// TIA Portal project "LVT_ModbusDeviceRtu_slow-poll_v0.0.1" (V17)

(* hardware
DEVICE "S7-1200 station_1"  S7-1200 Station
   slot 0: "Rack_0"  S7-1200 Rack  Rack  V1.0
   slot 1: "PLC_1"  CPU 1214C DC/DC/DC  6ES7 214-1AG40-0XB0  V4.3
   slot 3: "CB1"  CB 1241 (RS485)  6ES7 241-1CH30-1XB0  V1.0
*)

// ===== PLC "PLC_1"  CPU 1214C DC/DC/DC =====

VAR_GLOBAL   // PLC tag table "Default tag table"
   "System_Byte" AT %MB500 : Byte;
   "FirstScan" AT %M500.0 : Bool;
   "DiagStatusUpdate" AT %M500.1 : Bool;
   "AlwaysTRUE" AT %M500.2 : Bool;
   "AlwaysFALSE" AT %M500.3 : Bool;
   "System_Byte(1)" AT %MB1 : Byte;
   "System_Byte(2)" AT %MB1 : Byte;
   "Clock_Byte" AT %MB501 : Byte;
   "Clock_10Hz" AT %M501.0 : Bool;
   "Clock_5Hz" AT %M501.1 : Bool;
   "Clock_2.5Hz" AT %M501.2 : Bool;
   "Clock_2Hz" AT %M501.3 : Bool;
   "Clock_1.25Hz" AT %M501.4 : Bool;
   "Clock_1Hz" AT %M501.5 : Bool;
   "Clock_0.625Hz" AT %M501.6 : Bool;
   "Clock_0.5Hz" AT %M501.7 : Bool;
END_VAR

// folder: Example

TYPE "DeviceData"
   STRUCT
      param1 : Word;   // Parameter 1
      error : Bool;   // Flag. The device don't respond
   END_STRUCT;
END_TYPE

// folder: LVT_ModbusDeviceRtu

TYPE "LVT_typeModbusDeviceRtu_RequestCfg"
// Modbus request configuration
   STRUCT
      mode : USInt := 0;   // Mode / Режим опроса
      dataAddr : UDInt := 40001;   // Starting address in the slave / Начальный адрес регистра
      len : UInt := 1;   // Data length / Длина запроса
      mapAddr : DInt := 0;   // Starting address in the read/write buffer
      enable : Bool := false;   // Заблокировать запрос / Enable request
   END_STRUCT;
END_TYPE

TYPE "LVT_typeModbusDeviceRtu_Request"
   STRUCT
      cfg : "LVT_typeModbusDeviceRtu_RequestCfg";
      status : "LVT_typeModbusDeviceRtu_RequestStatus";
   END_STRUCT;
END_TYPE

TYPE "LVT_typeModbusDeviceRtu_Data"
   STRUCT
      address : UInt;   // Modbus RTU station address
      buffer : Array[0..100] of Word;   // Local buffer
      requests : Array[0..9] of "LVT_typeModbusDeviceRtu_Request";   // Requests
   END_STRUCT;
END_TYPE

TYPE "LVT_typeModbusDeviceRtu_RequestStatus"
// Modbus request status
   STRUCT
      req : Bool;   // Команда на отпарвку запроса / Send request
      done : Bool;   // Опрос завершен / Request is done
      busy : Bool;   // Блок в работе / Request is in progress
      error : Bool;   // Ошибка / Error
      status : Word;   // Статус / Error code
      errorCounter : UInt;   // Counter of failed attempts
   END_STRUCT;
END_TYPE

TYPE "LVT_typeModbusDeviceRtu_ComPortData"
TITLE = Настройки COM-порта
// Настройки COM-порта
   STRUCT
      port : Port := 271;   // ID порта / ID Port
      baud : UDInt := 9600;   // Скорость / Baudrate
      parity : UInt := 2;   // Паритет (0 - Нет, 1 - Нечет, 2 - Чет ) / Parity (0- None, 1 - Odd, 2 - Even)
      stopBits : UInt;   // Number of stop bits per character Valid values 1 and 2
      timeout : UInt := 500;   // Максимальное время ответа / Response timeout, ms
      retries : Word := 2;   // Количество повторных запросово / The number of repeated attempts by the master before the error code 0x80C8 is returned for "No response
      status : Word;   // Статус / Error codes
      done : Bool;   // Инициализация завершена / Execution of instruction completed without error
      error : Bool;   // Ошибка инициализации / Error
   END_STRUCT;
END_TYPE

// folder: Example/Data

DATA_BLOCK "DataDb"   // DB1
{ S7_Optimized_Access := 'TRUE' }
VERSION : 0.1
   VAR
      devices : Array[0..2] of "DeviceData";
   END_VAR
BEGIN
END_DATA_BLOCK

DATA_BLOCK "ModbusRtuMaster_DevicesDb"   // DB2
{ S7_Optimized_Access := 'TRUE' }
VERSION : 0.1
   VAR RETAIN
      devices : Array[0..2] of "LVT_typeModbusDeviceRtu_Data";
   END_VAR
BEGIN
   devices[0].address := 1;
   devices[1].address := 2;
   devices[2].address := 3;
   devices[0].requests[0].cfg.mode := 0;
   devices[0].requests[0].cfg.dataAddr := 40001;
   devices[0].requests[0].cfg.len := 1;
   devices[0].requests[0].cfg.mapAddr := 0;
   devices[0].requests[0].cfg.enable := true;
   devices[1].requests[0].cfg.mode := 0;
   devices[1].requests[0].cfg.dataAddr := 40001;
   devices[1].requests[0].cfg.len := 1;
   devices[1].requests[0].cfg.mapAddr := 0;
   devices[1].requests[0].cfg.enable := true;
   devices[2].requests[0].cfg.mode := 0;
   devices[2].requests[0].cfg.dataAddr := 40001;
   devices[2].requests[0].cfg.len := 1;
   devices[2].requests[0].cfg.mapAddr := 0;
   devices[2].requests[0].cfg.enable := true;
END_DATA_BLOCK

DATA_BLOCK "LVT_ModbusDeviceRtu_CfgDb"   // DB21
{ S7_Optimized_Access := 'TRUE' }
AUTHOR : Veshtemov
VERSION : 0.1
// Конфигурация регистров чтения по Modbus RTU
   VAR RETAIN
      com : "LVT_typeModbusDeviceRtu_ComPortData";
   END_VAR
BEGIN
   com.retries := 1;
   com.timeout := 500;
   com.port := 271;
   com.baud := 9600;
   com.parity := 0;
   com.stopBits := 0;
END_DATA_BLOCK

DATA_BLOCK "LVT_ModbusDeviceRtu_DataDb"   // DB24
{ S7_Optimized_Access := 'FALSE' }
VERSION : 0.1
   VAR
      readBuffer : Array[0..255] of Byte;
      writeBuffer : Array[0..255] of Byte;
   END_VAR
BEGIN
END_DATA_BLOCK

// folder: Example/Inst

DATA_BLOCK "inst_ModbusRtu_Master"   // DB3
{ S7_Optimized_Access := 'TRUE' }
VERSION : 0.1
// stored: InstanceOfName ModbusRtu_Master
"ModbusRtu_Master"
BEGIN
END_DATA_BLOCK

// folder: Example

ORGANIZATION_BLOCK "Main"   // OB1, SCL, ProgramCycle
TITLE = "Main Program Sweep (Cycle)"
{ S7_Optimized_Access := 'TRUE' }
VERSION : 0.1
   VAR_INPUT
      Initial_Call : Bool;   // Initial call of this OB
      Remanence : Bool;   // =True, if remanent data are available
   END_VAR
BEGIN
   "inst_ModbusRtu_Master"(com:="LVT_ModbusDeviceRtu_CfgDb".com,
                           mbCommLoad:="Modbus_Comm_Load_DB",
                           mbMaster:="Modbus_Master_DB");
END_ORGANIZATION_BLOCK

// folder: Example/RS485/ModbusRtuMaster

FUNCTION_BLOCK "ModbusRtu_Master"   // FB5, SCL
{ S7_Optimized_Access := 'TRUE' }
VERSION : 0.1
// Modbus Rtu Bus
   VAR_IN_OUT
      com : "LVT_typeModbusDeviceRtu_ComPortData";   // Serial port settings
      mbCommLoad : Modbus_Comm_Load;   // Instance of "Modbus_Comm_Load" function block
      mbMaster : Modbus_Master;   // Instance of "Modbus_Master" function block
   END_VAR
   VAR
      allowPolles : Array[0..#MAX_DEV_INDEX] of Bool;   // Allow polling
      slowPollTimers : Array[0..#MAX_DEV_INDEX] of TON_TIME;   // Slow poll timer
      stat_InitTrig : R_TRIG;   // Trig to set serial port is ready
      stat_LModbusDeviceRtu_Master : "LVT_ModbusDeviceRtu_Master";   // Instance of "LMBMD_ModbusDevice"
      i : Int := 0;   // Index
      j : Int := 0;   // Index
      statStart : Bool;   // Flag to start polling
   END_VAR
   VAR CONSTANT
      MAX_DEV_INDEX : Int := 2;   // Max index in devices array
      SLOW_POLL_TIME : Time := T#10s;   // Slow poll time
   END_VAR
BEGIN
   REGION Block info header
       //===============================================================================
       // (company) / (c)Copyright year
       //-------------------------------------------------------------------------------
       // Title:            Example of LVT _ModbusDevcieRtu library
       // Comment/Function: Modbus RTU Master device-oriented
       //                   This functional block polls 1 register in 3 indentical devices,
       //                   If a device fails to respond 3 times, a slowPollTimer is activated 
       //                   and polling is blocked until timer expires
       // Library/Family:   LMB (Library Modbus)
       // Author:           Anatoly Veshtemov
       // Tested with:      CPU 1214C
       // Engineering:      TIA Portal V17
       // Restrictions:     no
       // Requirements:     PLC (S7-1200 / S7-1500)
       //-------------------------------------------------------------------------------
       // Change log table:
       // Version  | Date       | Expert in charge       | Changes applied
       //----------|------------|------------------------|------------------------------
       // 00.01.00 17.06.2026  First release
       //=============================================================================

   END_REGION Block info header

   REGION DESCRIPTION
       (/**/)
   END_REGION DESCRIPTION


   // Modbus RTU Master

   REGION Serial port initialization
       IF "FirstScan" THEN
           #mbCommLoad.MODE := 4;
       END_IF;

       #mbCommLoad.RETRIES := #com.retries;

       #mbCommLoad(REQ := "FirstScan",
                   "PORT" := #com."port",
                   BAUD := #com.baud,
                   PARITY := #com.parity,
                   MB_DB := #mbMaster.MB_DB,
                   RESP_TO := #com.timeout,
                   DONE => #com.done,
                   ERROR => #com.error,
                   STATUS => #com.status);

       #stat_InitTrig(CLK := #com.done);

       IF #stat_InitTrig.Q THEN
           #i := 0;
       END_IF;
   END_REGION

   #statStart := NOT #stat_LModbusDeviceRtu_Master.done;

   REGION Slow poll

       FOR #j := 0 TO #MAX_DEV_INDEX DO

           // Update Slow Poll timers
           #slowPollTimers[#j](IN := "DataDb".devices[#j].error,
                               PT := #SLOW_POLL_TIME);

           // Polling is allowed if there are no error or timer is ended.        
           #allowPolles[#j] := NOT ("DataDb".devices[#j].error AND #slowPollTimers[#j].Q);

       END_FOR;

   END_REGION

   CASE #i OF
       0..#MAX_DEV_INDEX:  // Device 1..Devices 3

           IF #allowPolles[#i] THEN
               #stat_LModbusDeviceRtu_Master(start := #statStart,
                                             readBuffer := "LVT_ModbusDeviceRtu_DataDb".readBuffer,
                                             writeBuffer := "LVT_ModbusDeviceRtu_DataDb".writeBuffer,
                                             data := "ModbusRtuMaster_DevicesDb".devices[#i],
                                             mbMaster := #mbMaster);

               IF #stat_LModbusDeviceRtu_Master.done THEN

                   "ModbusRtu_Device_HandleData"(mdata := "ModbusRtuMaster_DevicesDb".devices[#i],
                                                 data := "DataDb".devices[#i]);

                   #i := #i + 1;
               END_IF;

           ELSE
               #i := #i + 1;
           END_IF;

       ELSE
           #i := 0;
   END_CASE;
END_FUNCTION_BLOCK

FUNCTION "ModbusRtu_Device_HandleData" : Void   // FC18, SCL
{ S7_Optimized_Access := 'TRUE' }
VERSION : 0.1
   VAR_IN_OUT
      mdata : "LVT_typeModbusDeviceRtu_Data";
      data : "DeviceData";
   END_VAR
   VAR_TEMP
      i : Int;   // Increment
      statQuantityErrors : UInt;   // Quantity of failed requests
   END_VAR
   VAR CONSTANT
      ERRORS_THRESHOLD : Int := 3;   // Max. quantity of failed requests
      MAX_REQUEST_INDEX : Int := 9;   // Max. index of array with requests
   END_VAR
BEGIN
   REGION Block info header
       //===============================================================================
       // (company) / (c)Copyright year
       //-------------------------------------------------------------------------------
       // Title:            Example of LVT_ModbusDevcieRtu library
       // Comment/Function: Modbus RTU Master device-oriented
       //                   Copy data to device from modbus buffer, set connection status
       // Library/Family:   LVT 
       // Author:           Anatoly Veshtemov
       // Tested with:      CPU 1214C
       // Engineering:      TIA Portal V17
       // Restrictions:     no
       // Requirements:     PLC (S7-1200 / S7-1500)
       //-------------------------------------------------------------------------------
       // Change log table:
       // Version  | Date       | Expert in charge       | Changes applied
       //----------|------------|------------------------|------------------------------
       // 00.00.01 17.06.2026  First release
       //=============================================================================

   END_REGION Block info header

   REGION DESCRIPTION
       (/**/)
   END_REGION DESCRIPTION


   // Data
   #data.param1 := #mdata.buffer[0];

   // Calculate quantity of failed requests
   #statQuantityErrors := 0;
   FOR #i := 0 TO #MAX_REQUEST_INDEX - 1 DO
       #statQuantityErrors += #mdata.requests[#i].status.errorCounter;
   END_FOR;

   // Set error status
   #data.error := #statQuantityErrors >= #ERRORS_THRESHOLD;
END_FUNCTION

// folder: LVT_ModbusDeviceRtu

FUNCTION "LVT_ModbusDeviceRtu_Description" : Void   // FC3, SCL
{ S7_Optimized_Access := 'TRUE' }
AUTHOR : Anatoly Veshtemov
FAMILY : LVT
BEGIN
   REGION INFO
   (/*title: Library for Modbus Rtu Master
   subTitle: STEP 7 Basic/Professional (TIA PORTAL) / SIMATIC S7-1200 / S7-1500
   shortDescription: Modbus RTU Master device-oriented library for S7-1200/S7-1500
   type: Library
   fileName: LVT_ModbusDeviceRtu_Lib
   link: https://github.com/vapik/simatic-modbus-device-master*/)
   END_REGION INFO

   REGION ChangeLog
   (*
   Version  | Date       | Expert in charge       | Changes applied
   ---------|------------|------------------------|------------------------------
   00.01.00 | 17.06.2026 | Upgrate to TIA V17
            |            | Added block info headers
            |            | Refactor names
            |            | Examples has deleted                  
            |            | Chanhed name to LVT_ModbusDeviceRtu                           
   *)
   END_REGION
END_FUNCTION

// folder: LVT_ModbusDeviceRtu/Core

FUNCTION_BLOCK "LVT_ModbusDeviceRtu_Master"   // FB7, SCL
{ S7_Optimized_Access := 'TRUE' }
AUTHOR : Anatoly Veshtemov
FAMILY : LVT
   VAR_INPUT
      start : Bool;   // Пуск / Start block
   END_VAR
   VAR_OUTPUT
      busy : Bool;   // В процессе / In progress
      done : Bool;   // Окончание / Done
   END_VAR
   VAR_IN_OUT
      readBuffer : Variant;   // Буфер обмена / Pointer of read buffer (non optimized data block). For example, DB -> readBuffer: Array[0..125] of Word
      writeBuffer : Variant;   // Pointer of write buffer (non optimized data block). For example, DB -> writeBuffer: Array[0..125] of Word
      data : "LVT_typeModbusDeviceRtu_Data";
      mbMaster : Modbus_Master;   // Instance of Modbus_Master function block
   END_VAR
   VAR
      statBuffer : Array[0..127] of Word;
      startTrig : R_TRIG;   // Detect start
      statWatchdogTimer : TON_TIME;   // Timer for resetting a request when unknown reason is happened
      statState : USInt;   // Текущая стадия обмена / Current state
      i : Int;
      j : Int;
   END_VAR
   VAR_TEMP
      tempStart : Bool;   // Start flag
      tempRetval : Int;
      tempQntRequests : Int;   // Quantity of requests
      tempZeroIndex : DInt;
   END_VAR
   VAR CONSTANT
      STATE_STANDBY : USInt := 0;   // Ожидание / State. Standby
      STATE_SETTINGS : USInt := 1;   // Конфигурирование запроса / State. Get settings
      STATE_READ : USInt := 2;   // Запрос на чтение / State. Reading
      STATE_WRITE : USInt := 3;   // Запрос на запись / State. Writing
      STATE_HANDLE : USInt := 4;   // Обработка запроса / State. Handle results
      WATCHDOG_TIME : Time := T#10S;   // Максимальное время ожидания / Watchdog time
      ERROR_ILLEGAL_REQUEST : Word := 16#9000;   // Error. Illegal request (check request settings)
      ERROR_WATCHDOG_TIMER : Word := 16#9001;   // Error. Watchdog timer
   END_VAR
BEGIN
   REGION Block info header
       //===============================================================================
       // (company) / (c)Copyright year
       //-------------------------------------------------------------------------------
       // Title:            LVT_ModbusDevcieRtu_Master
       // Comment/Function: Modbus RTU Master device-oriented
       //                   Requests are grouped for each network device separately, and devices are sequentially polled.
       //                   Each network device has a local data buffer.
       // Library/Family:   LVT
       // Author:           Anatoly Veshtemov
       // Tested with:      CPU 1214C
       // Engineering:      TIA Portal V17
       // Restrictions:     no
       // Requirements:     PLC (S7-1200 / S7-1500)
       //-------------------------------------------------------------------------------
       // Change log table:
       // Version  | Date       | Expert in charge       | Changes applied
       //----------|------------|------------------------|------------------------------
       // 00.00.04 01.01.2023  First released version
       // 00.01.00 17.06.2026  Upgrate to TIA V17
       //                      Added block info header
       //                      Refactor names in Static 
       //=============================================================================

   END_REGION Block info header

   REGION DESCRIPTION
       (/**/)
   END_REGION DESCRIPTION

   #tempQntRequests := UDINT_TO_INT("LVT_ModbusDeviceRtu_GetArrayLength"(arr := #data.requests));
   #busy := (#statState > #STATE_STANDBY); // Set busy flag

   #startTrig(CLK := #start,
                   Q => #tempStart);

   // When start go to Settings
   IF #tempStart THEN

       #done := false;
       #statState := #STATE_SETTINGS;

   END_IF;

   CASE #statState OF

           // Standby
       #STATE_STANDBY:

           #done := false;
           #i := 0;

           // Get request settings
       #STATE_SETTINGS:

           // With the first call we reset the counter, get the first request,
           // else we increase counter by 1 and get a next request
           IF #tempStart THEN
               #i := 0;

           ELSE
               #i := #i + 1;

               // When all requests is completed go to standby, set "done" flag 
               IF #i >= #tempQntRequests THEN
                   #done := true;
                   #statState := #STATE_STANDBY;
                   RETURN;
               END_IF;
           END_IF;

           // Check request settings: we have to skip disabled or invalid requests,
           // if a request is invalid - set ERROR_ILLEGAL_REQUEST status
           FOR #j := #i TO #tempQntRequests - 1 DO

               IF NOT #data.requests[#j].cfg.enable THEN

                   #data.requests[#j].status.req := false;
                   #data.requests[#j].status.done := false;
                   #data.requests[#j].status.error := false;
                   #data.requests[#j].status.status := 0;
                   #data.requests[#j].status.errorCounter := 0;

               ELSIF NOT "LVT_ModbusDeviceRtu_ValidateRequest"(data := #data, index := #j) THEN

                   // Set error status
                   #data.requests[#j].status.req := false;
                   #data.requests[#j].status.done := false;
                   #data.requests[#j].status.error := true;
                   #data.requests[#j].status.status := #ERROR_ILLEGAL_REQUEST;
                   #data.requests[#j].status.errorCounter := LIMIT(IN := #data.requests[#j].status.errorCounter + 1,
                                                                   MN := 0,
                                                                   MX := 65534);
               ELSE
                   #i := #j;
                   EXIT;
               END_IF;

               // When all requests is completed go to standby, set "done" flag
               IF #j = #tempQntRequests - 1 THEN
                   #done := true;
                   #statState := #STATE_STANDBY;
                   RETURN;
               END_IF;

           END_FOR;

           // For writing before request we have to copy data to external write buffer
           IF #data.requests[#i].cfg.mode > 0 THEN

               // Extract data from Modbus Device to write buffer
               MOVE_BLK(IN := #data.#buffer[#data.requests[#i].cfg.mapAddr],
                        COUNT := #data.requests[#i].cfg.len,
                        OUT => #statBuffer[0]);

               #tempZeroIndex := 0;
               #tempRetval := Serialize(SRC_VARIABLE := #statBuffer,
                                        DEST_ARRAY => #writeBuffer,
                                        POS := #tempZeroIndex);

               #statState := #STATE_WRITE;
           ELSE
               #statState := #STATE_READ;
           END_IF;

           RETURN;

           // Read
       #STATE_READ, #STATE_WRITE:

           #data.requests[#i].status.req := true;

           // Handle results
       #STATE_HANDLE:

           #data.requests[#i].status.req := false;

           IF #data.requests[#i].status.done THEN
               #data.requests[#i].status.errorCounter := 0;

               // Copy from modbus buffer to device buffer
               IF #data.requests[#i].cfg.mode = 0 THEN

                   #tempZeroIndex := 0;
                   #tempRetval := Deserialize(SRC_ARRAY := #readBuffer,
                                              DEST_VARIABLE => #statBuffer,
                                              POS := #tempZeroIndex);
                   MOVE_BLK(IN := #statBuffer[0],
                            COUNT := #data.requests[#i].cfg.len,
                            OUT => #data.buffer[#data.requests[#i].cfg.mapAddr]);
               END_IF;

           ELSIF #data.requests[#i].status.error THEN
               #data.requests[#i].status.errorCounter := LIMIT(IN := #data.requests[#i].status.errorCounter + 1,
                                                               MN := 0,
                                                               MX := 65534);
           END_IF;

           #statState := #STATE_SETTINGS;

       ELSE
           #statState := #STATE_STANDBY;
   END_CASE;

   // There are different buffers for reading and writing
   IF (#statState = #STATE_READ) THEN
       // Request
       #mbMaster(REQ := #data.requests[#i].status.req,
                 MB_ADDR := #data.address,
                 MODE := #data.requests[#i].cfg.mode,
                 DATA_ADDR := #data.requests[#i].cfg.dataAddr,
                 DATA_LEN := #data.requests[#i].cfg.len,
                 DONE => #data.requests[#i].status.done,
                 BUSY => #data.requests[#i].status.busy,
                 ERROR => #data.requests[#i].status.error,
                 STATUS => #data.requests[#i].status.status,
                 DATA_PTR := #readBuffer);

   ELSIF (#statState = #STATE_WRITE) THEN
       // Request
       #mbMaster(REQ := #data.requests[#i].status.req,
                 MB_ADDR := #data.address,
                 MODE := #data.requests[#i].cfg.mode,
                 DATA_ADDR := #data.requests[#i].cfg.dataAddr,
                 DATA_LEN := #data.requests[#i].cfg.len,
                 DONE => #data.requests[#i].status.done,
                 BUSY => #data.requests[#i].status.busy,
                 ERROR => #data.requests[#i].status.error,
                 STATUS => #data.requests[#i].status.status,
                 DATA_PTR := #writeBuffer);
   END_IF;


   // Waiting response status
   IF ((#statState = #STATE_READ
       OR #statState = #STATE_WRITE)
       AND (#data.requests[#i].status.done
       OR #data.requests[#i].status.error))
   THEN
       #statState := #STATE_HANDLE;
   END_IF;

   // Watchdog timer is needed when state stuck in Read or Write state for unknown reason,
   // in that case we set request as invalid 
   #statWatchdogTimer(IN := (#statState = #STATE_READ
                       OR #statState = #STATE_WRITE),
                       PT := #WATCHDOG_TIME);

   IF #statWatchdogTimer.Q THEN

       #data.requests[#i].status.done := false;
       #data.requests[#i].status.error := true;
       #data.requests[#i].status.status := #ERROR_WATCHDOG_TIMER;
       #data.requests[#i].status.errorCounter := LIMIT(IN := #data.requests[#i].status.errorCounter + 1,
                                                       MN := 0,
                                                       MX := 65534);

       #statState := #STATE_HANDLE;

   END_IF;
END_FUNCTION_BLOCK

FUNCTION "LVT_ModbusDeviceRtu_ValidateRequest" : Bool   // FC2, SCL
{ S7_Optimized_Access := 'TRUE' }
AUTHOR : Anatoly Veshtemov
FAMILY : LVT
   VAR_INPUT
      index : Int;   // Index of request
   END_VAR
   VAR_IN_OUT
      data : "LVT_typeModbusDeviceRtu_Data";
   END_VAR
   VAR_TEMP
      tempBufferSize : Int;   // Size of data.buffer
   END_VAR
BEGIN
   REGION Block info header
       //===============================================================================
       // (company) / (c)Copyright year
       //-------------------------------------------------------------------------------
       // Title:            LVT_ModbusDevcieRtu_Master
       // Comment/Function: Modbus RTU Master device-oriented
       //                   Check settings of request: valid length, mode and mapping

       // Library/Family:   LVT 
       // Author:           Anatoly Veshtemov
       // Tested with:      CPU 1214C
       // Engineering:      TIA Portal V17
       // Restrictions:     no
       // Requirements:     PLC (S7-1200 / S7-1500)
       //-------------------------------------------------------------------------------
       // Change log table:
       // Version  | Date       | Expert in charge       | Changes applied
       //----------|------------|------------------------|------------------------------
       // 00.00.04 01.01.2023  First released version
       // 00.01.00 17.06.2026  Upgrate to TIA V17
       //                      Added block info header
       //=============================================================================

   END_REGION Block info header

   REGION DESCRIPTION
       (/**/)
   END_REGION DESCRIPTION

   #tempBufferSize := UDINT_TO_INT("LVT_ModbusDeviceRtu_GetArrayLength"(arr := #data.buffer));

   // Check request:
   // * Valid length
   // * Valid mode
   // * Valid mapping to/from buffer
   // other will be checking by Modbus_Master FB

   #LVT_ModbusDeviceRtu_ValidateRequest :=
   #data.requests[#index].cfg.len > 0
   AND (#data.requests[#index].cfg.mode >= 0 AND #data.requests[#index].cfg.mode <= 2)
   AND (#data.requests[#index].cfg.mapAddr + #data.requests[#index].cfg.len) <= #tempBufferSize
   ;
END_FUNCTION

FUNCTION "LVT_ModbusDeviceRtu_GetArrayLength" : UDInt   // FC9, SCL
{ S7_Optimized_Access := 'TRUE' }
AUTHOR : Anatoly Veshtemov
FAMILY : LVT
   VAR_INPUT
      arr : Variant;
   END_VAR
BEGIN
   REGION Block info header
       //===============================================================================
       // (company) / (c)Copyright year
       //-------------------------------------------------------------------------------
       // Title:            LVT_ModbusDevcieRtu_Master
       // Comment/Function: Modbus RTU Master device-oriented
       //                   Get array length
       // Library/Family:   LVT
       // Author:           Anatoly Veshtemov
       // Tested with:      CPU 1214C
       // Engineering:      TIA Portal V17
       // Restrictions:     no
       // Requirements:     PLC (S7-1200 / S7-1500)
       //-------------------------------------------------------------------------------
       // Change log table:
       // Version  | Date       | Expert in charge       | Changes applied
       //----------|------------|------------------------|------------------------------
       // 00.00.04 01.01.2023  First released version
       //=============================================================================

   END_REGION Block info header

   REGION DESCRIPTION
       (/**/)
   END_REGION DESCRIPTION

   IF IS_ARRAY(#arr) THEN
       #LVT_ModbusDeviceRtu_GetArrayLength := CountOfElements(IN := #arr);
   ELSE
       #LVT_ModbusDeviceRtu_GetArrayLength := 0;
   END_IF;
END_FUNCTION

// ===== library: MasterCopy "LMB_ModbusDeviceRtu_Buffer" =====

// folder: LMB_ModbusDeviceRtu_Master

TYPE "LMB_ModbusDeviceRtu_Buffer"
// Raw data of Modbus device
   STRUCT
      readBuffer : Array[0..100] of Word;   // Read buffer
      writeBuffer : Array[0..100] of Word;   // Write buffer
   END_STRUCT;
END_TYPE

// ===== library: MasterCopy "LMB_ModbusDeviceRtu_ComPortData" =====

// folder: LMB_ModbusDeviceRtu_Master

TYPE "LMB_ModbusDeviceRtu_ComPortData"
TITLE = Настройки COM-порта
// Настройки COM-порта
   STRUCT
      port : Port := 271;   // ID порта / ID Port
      baud : UDInt := 9600;   // Скорость / Baudrate
      parity : UInt := 2;   // Паритет (0 - Нет, 1 - Нечет, 2 - Чет ) / Parity (0- None, 1 - Odd, 2 - Even)
      stopBits : UInt;   // Number of stop bits per character Valid values 1 and 2
      timeout : UInt := 500;   // Максимальное время ответа / Response timeout, ms
      status : Word;   // Статус / Response timeout
      done : Bool;   // Инициализация завершена / Execution of instruction completed without error
      error : Bool;   // Ошибка инициализации / Error
      retries : Word := 2;   // Количество повторных запросово / The number of repeated attempts by the master before the error code 0x80C8 is returned for "No response
   END_STRUCT;
END_TYPE

// ===== library: MasterCopy "LMB_ModbusDeviceRtu_Data" =====

// folder: LMB_ModbusDeviceRtu_Master

TYPE "LMB_ModbusDeviceRtu_Data"
   STRUCT
      addresss : UInt;   // Modbus RTU station address
      buffer : "LMB_ModbusDeviceRtu_Buffer";
      requests : Array[0..9] of "LMB_ModbusDeviceRtu_Request";
   END_STRUCT;
END_TYPE

// ===== library: MasterCopy "LMB_ModbusDeviceRtu_Request" =====

// folder: LMB_ModbusDeviceRtu_Master

TYPE "LMB_ModbusDeviceRtu_Request"
   STRUCT
      cfg : "LMB_ModbusDeviceRtu_RequestCfg";
      status : "LMB_ModbusDeviceRtu_RequestStatus";
   END_STRUCT;
END_TYPE

// ===== library: MasterCopy "LMB_ModbusDeviceRtu_RequestCfg" =====

// folder: LMB_ModbusDeviceRtu_Master

TYPE "LMB_ModbusDeviceRtu_RequestCfg"
// Modbus request configuration
   STRUCT
      mode : USInt := 0;   // Mode / Режим опроса
      dataAddr : UDInt := 40001;   // Starting address in the slave / Начальный адрес регистра
      len : UInt := 1;   // Data length / Длина запроса
      mapAddr : DInt := 0;   // Starting address in the read/write buffer
      enable : Bool := false;   // Заблокировать запрос / Enable request
   END_STRUCT;
END_TYPE

// ===== library: MasterCopy "LMB_ModbusDeviceRtu_RequestStatus" =====

// folder: LMB_ModbusDeviceRtu_Master

TYPE "LMB_ModbusDeviceRtu_RequestStatus"
// Modbus request status
   STRUCT
      req : Bool;   // Команда на отпарвку запроса
      done : Bool;   // Опрос завершен
      busy : Bool;   // Блок в работе
      error : Bool;   // Ошибка
      status : Word;   // Статус / Error code
      errorCounter : UInt;
   END_STRUCT;
END_TYPE

// ===== library: MasterCopy "LMB_ModbusDeviceRtu_GetArrayLength" =====

// folder: LMB_ModbusDeviceRtu_Master/Core

FUNCTION "LMB_ModbusDeviceRtu_GetArrayLength" : UDInt   // FC9, SCL
{ S7_Optimized_Access := 'TRUE' }
VERSION : 0.1
   VAR_INPUT
      arr : Variant;
   END_VAR
BEGIN
   IF IS_ARRAY(#arr) THEN
       #LMB_ModbusDeviceRtu_GetArrayLength := CountOfElements(IN := #arr);
   ELSE
       #LMB_ModbusDeviceRtu_GetArrayLength := 0;
   END_IF;
END_FUNCTION

// ===== library: MasterCopy "LMB_ModbusDeviceRtu_ValidateRequest" =====

// folder: LMB_ModbusDeviceRtu_Master/Core

FUNCTION "LMB_ModbusDeviceRtu_ValidateRequest" : Bool   // FC2, SCL
{ S7_Optimized_Access := 'TRUE' }
VERSION : 0.1
   VAR_IN_OUT
      data : "LMB_ModbusDeviceRtu_RequestCfg";
   END_VAR
BEGIN
   #LMB_ModbusDeviceRtu_ValidateRequest :=
   #data.len > 0
   AND (#data.mode >= 0 AND #data.mode <= 2);
END_FUNCTION

// ===== library: MasterCopy "LMB_ModbusDeviceRtu_Master" =====

// folder: LMB_ModbusDeviceRtu_Master/Core

FUNCTION_BLOCK "LMB_ModbusDeviceRtu_Master"   // FB7, SCL
{ S7_Optimized_Access := 'TRUE' }
VERSION : 0.1
   VAR_INPUT
      start : Bool;   // Пуск / Start block
   END_VAR
   VAR_OUTPUT
      busy : Bool;   // В процессе / In progress
      done : Bool;   // Окончание / Done
   END_VAR
   VAR_IN_OUT
      readBuffer : Variant;   // Буфер обмена / Pointer of read buffer (non optimized data block). For example, DB -> readBuffer: Array[0..125] of Word
      writeBuffer : Variant;   // Pointer of write buffer (non optimized data block). For example, DB -> writeBuffer: Array[0..125] of Word
      data : "LMB_ModbusDeviceRtu_Data";
      mbMaster : Modbus_Master;   // Instance of Modbus_Master function block
   END_VAR
   VAR
      inst_startTrig : R_TRIG;   // Detect start
      inst_watchdogTimer : TON_TIME;   // Timer for resetting a request when unknown reason is happened
      state : USInt;   // Текущая стадия обмена / Current state
      i : Int;
      j : Int;
   END_VAR
   VAR_TEMP
      tempStart : Bool;   // Start flag
      tempRetval : Int;
      tempQntRequests : Int;   // Quantity of requests
   END_VAR
   VAR CONSTANT
      STATE_STANDBY : USInt := 0;   // Ожидание / State. Standby
      STATE_SETTINGS : USInt := 1;   // Конфигурирование запроса / State. Get settings
      STATE_READ : USInt := 2;   // Запрос на чтение / State. Reading
      STATE_WRITE : USInt := 3;   // Запрос на запись / State. Writing
      STATE_HANDLE : USInt := 4;   // Обработка запроса / State. Handle results
      WATCHDOG_TIME : Time := T#10S;   // Максимальное время ожидания / Watchdog time
      ERROR_ILLEGAL_REQUEST : Word := 16#8500;   // Error. Illegal request (check request settings)
      ERROR_WATCHDOG_TIMER : Word := 16#8501;   // Error. Watchdog timer
   END_VAR
BEGIN
   #tempQntRequests := UDINT_TO_INT("LMB_ModbusDeviceRtu_GetArrayLength"(arr := #data.requests));
   #busy := (#state > #STATE_STANDBY); // Set busy flag

   #inst_startTrig(CLK := #start, Q => #tempStart);

   // When start go to Settings
   IF #tempStart THEN

       #done := false;
       #state := #STATE_SETTINGS;

   END_IF;

   CASE #state OF

       // Standby
       #STATE_STANDBY:

           #done := false;
           #i := 0;

       // Get request settings
       #STATE_SETTINGS:

           // With the first call we reset the counter, get the first request,
           // else we increase counter by 1 and get a next request
           IF #tempStart THEN
               #i := 0;

           ELSE
               #i := #i + 1;

               // When all requests is completed go to standby, set "done" flag 
               IF #i >= #tempQntRequests THEN
                   #done := true;
                   #state := #STATE_STANDBY;
                   RETURN;
               END_IF;
           END_IF;

           // Check request settings: we have to skip disabled or invalid requests,
           // if a request is invalid - set ERROR_ILLEGAL_REQUEST status
           FOR #j := #i TO #tempQntRequests - 1 DO

               IF NOT #data.requests[#j].cfg.enable THEN

                   #data.requests[#j].status.req := false;
                   #data.requests[#j].status.done := false;
                   #data.requests[#j].status.error := false;
                   #data.requests[#j].status.status := 0;
                   #data.requests[#j].status.errorCounter := 0;

               ELSIF NOT "LMB_ModbusDeviceRtu_ValidateRequest"(#data.requests[#j].cfg) THEN

                   // Set error status
                   #data.requests[#j].status.req := false;
                   #data.requests[#j].status.done := false;
                   #data.requests[#j].status.error := true;
                   #data.requests[#j].status.status := #ERROR_ILLEGAL_REQUEST;
                   #data.requests[#j].status.errorCounter := LIMIT(IN := #data.requests[#j].status.errorCounter + 1,
                                                                   MN := 0,
                                                                   MX := 65534);
               ELSE
                   #i := #j;
                   EXIT;
               END_IF;

               // When all requests is completed go to standby, set "done" flag
               IF #j = #tempQntRequests - 1 THEN
                   #done := true;
                   #state := #STATE_STANDBY;
                   RETURN;
               END_IF;

           END_FOR;

           // For writing before request we have to copy data to external write buffer
           IF #data.requests[#i].cfg.mode > 0 THEN

               // Extract data from Modbus Device write buffer
               #tempRetval := Serialize(SRC_VARIABLE := #data.buffer.writeBuffer,
                                        DEST_ARRAY => #writeBuffer,
                                        POS := #data.requests[#i].cfg.mapAddr);
               #state := #STATE_WRITE;
           ELSE
               #state := #STATE_READ;
           END_IF;

           RETURN;

       // Read
       #STATE_READ, #STATE_WRITE:

           #data.requests[#i].status.req := true;

       // Handle results
       #STATE_HANDLE:

           #data.requests[#i].status.req := false;

           IF #data.requests[#i].status.done THEN
               #data.requests[#i].status.errorCounter := 0;
           ELSIF #data.requests[#i].status.error THEN
               #data.requests[#i].status.errorCounter := LIMIT(IN := #data.requests[#i].status.errorCounter + 1,
                                                               MN := 0,
                                                               MX := 65534);
           END_IF;

           #state := #STATE_SETTINGS;

       ELSE
           #state := #STATE_STANDBY;
   END_CASE;

   // There are different buffers for reading and writing
   IF (#state = #STATE_READ) THEN
       // Request
       #mbMaster(REQ := #data.requests[#i].status.req,
                 MB_ADDR := #data.address,
                 MODE := #data.requests[#i].cfg.mode,
                 DATA_ADDR := #data.requests[#i].cfg.dataAddr,
                 DATA_LEN := #data.requests[#i].cfg.len,
                 DONE => #data.requests[#i].status.done,
                 BUSY => #data.requests[#i].status.busy,
                 ERROR => #data.requests[#i].status.error,
                 STATUS => #data.requests[#i].status.status,
                 DATA_PTR := #readBuffer);

   ELSIF (#state = #STATE_WRITE) THEN
       // Запрос
       #mbMaster(REQ := #data.requests[#i].status.req,
                 MB_ADDR := #data.address,
                 MODE := #data.requests[#i].cfg.mode,
                 DATA_ADDR := #data.requests[#i].cfg.dataAddr,
                 DATA_LEN := #data.requests[#i].cfg.len,
                 DONE => #data.requests[#i].status.done,
                 BUSY => #data.requests[#i].status.busy,
                 ERROR => #data.requests[#i].status.error,
                 STATUS => #data.requests[#i].status.status,
                 DATA_PTR := #writeBuffer);
   END_IF;


   // Waiting response status
   IF ((#state = #STATE_READ
       OR #state = #STATE_WRITE)
       AND (#data.requests[#i].status.done
       OR #data.requests[#i].status.error))
   THEN
       #state := #STATE_HANDLE;
   END_IF;

   // Watchdog timer is needed when state stuck in Read or Write state for unknown reason,
   // in that case we set request as invalid 
   #inst_watchdogTimer(IN := (#state = #STATE_READ
                  OR #state = #STATE_WRITE),
                  PT := #WATCHDOG_TIME);

   IF #inst_watchdogTimer.Q THEN

       #data.requests[#i].status.done := false;
       #data.requests[#i].status.error := true;
       #data.requests[#i].status.status := #ERROR_WATCHDOG_TIMER;
       #data.requests[#i].status.errorCounter := LIMIT(IN := #data.requests[#i].status.errorCounter + 1,
                                                       MN := 0,
                                                       MX := 65534);

       #state := #STATE_HANDLE;

   END_IF;
END_FUNCTION_BLOCK

// ===== library: MasterCopy "LMB_ModbusDeviceRtu_CfgDb" =====

// folder: LMB_ModbusDeviceRtu_Master/Data

DATA_BLOCK "LMB_ModbusDeviceRtu_CfgDb"   // DB21
{ S7_Optimized_Access := 'TRUE' }
AUTHOR : Veshtemov
VERSION : 0.1
// Конфигурация регистров чтения по Modbus RTU
   VAR
      com : "LMB_ModbusDeviceRtu_ComPortData";
   END_VAR
BEGIN
   com.port := 269;
   com.baud := 9600;
   com.retries := 1;
   com.parity := 2;
   com.stopBits := 1;
END_DATA_BLOCK

// ===== library: MasterCopy "LMB_ModbusDeviceRtu_DataDb" =====

// folder: LMB_ModbusDeviceRtu_Master/Data

DATA_BLOCK "LMB_ModbusDeviceRtu_DataDb"   // DB24
{ S7_Optimized_Access := 'FALSE' }
VERSION : 0.1
   VAR
      buffer : Array[0..125] of Word;
      writeBuffer : Array[0..125] of Word;
   END_VAR
BEGIN
END_DATA_BLOCK